FUNCTION_BLOCK FB_Homing_Direct EXTENDS FB_Homing_Base
VAR_INPUT
    ReferencePosition : LREAL := 0.0;
END_VAR
VAR
    fbMcHome          : MC_Home;
    fbMoveAbs         : MC_MoveAbsolute;
    DelayTimer        : TON;
	_HomingVelocity   : LREAL := 50.0;
END_VAR

METHOD Abort
VAR_INPUT
END_VAR
IF _Axis <> 0 THEN
    fbMcHome(Axis := _Axis.Axis, Execute := FALSE);
    fbMoveAbs(Axis := _Axis.Axis, Execute := FALSE);
END_IF

SUPER^.Abort();
END_METHOD

METHOD CyclicLogic
CASE nStep OF
    0: 
        fbMcHome(Axis := _Axis.Axis, Execute := FALSE);
        fbMoveAbs(Axis := _Axis.Axis, Execute := FALSE);

    10: 
        IF _Axis.Axis.Status.Homed THEN
            nStep := 20;
        ELSE
            fbMcHome(
                Axis        := _Axis.Axis, 
                Execute     := TRUE, 
                Position    := ReferencePosition,
                HomingMode  := MC_Direct
            );
            
            IF fbMcHome.Done THEN
                fbMcHome(Axis := _Axis.Axis, Execute := FALSE);
                nStep := 20;
            ELSIF fbMcHome.Error THEN
                _bBusy    := FALSE;
                _bError   := TRUE;
                _bErrorID := fbMcHome.ErrorID;
                nStep     := 0;
            END_IF
        END_IF

    20: 
        fbMoveAbs(
            Axis     := _Axis.Axis,
            Execute  := TRUE,
			Velocity := _HomingVelocity,
            Position := 0.0
        );
        
        IF fbMoveAbs.Done THEN
            fbMoveAbs(Axis := _Axis.Axis, Execute := FALSE);
            nStep := 40;
        ELSIF fbMoveAbs.Error THEN
            _bBusy    := FALSE;
            _bError   := TRUE;
            _bErrorID := fbMoveAbs.ErrorID;
            nStep     := 0;
        END_IF
        
    40: 
        _bBusy := FALSE;
        _bDone := TRUE; 
        nStep  := 0;
END_CASE
END_METHOD

PROPERTY HomingVelocity : LREAL
GET
HomingVelocity := _HomingVelocity;
END_GET
SET
_HomingVelocity := HomingVelocity;
END_SET
END_PROPERTY

END_FUNCTION_BLOCK

(* stored: Version 1.1.0.1, ProductVersion 3.1.4024.15
   POU FB_Homing_Direct: Id {9b95ef4f-a5ad-4500-8bd8-c009b6c64182}, SpecialFunc None
   Method Abort: Id {11112222-3333-4444-bbbb-111111111111}
   Method CyclicLogic: Id {22223333-4444-5555-bbbb-222222222222}
   Property HomingVelocity: Id {3f3d8927-9408-4cd7-a0bf-1a57402b1b16}
   Get Get: Id {c93d9d27-c57a-4121-985e-3d7fed3d16f5}
   Set Set: Id {5340dd65-c2c2-4f94-84b0-97558e14820f} *)
